// TwinCAT 3 PLC project PLC
// ProgramVersion: 3.1.4024.0
// libraries:
//   CmpBitmapPool, * (System)
//   Tc2_Standard, * (Beckhoff Automation GmbH)
//   Tc2_System, * (Beckhoff Automation GmbH)
//   Tc3_Module, * (Beckhoff Automation GmbH)
//   VisuDialogs, * (System)
//   VisuSymbols,3.5.10.0,System
// project tree:
//   DUTs/ DPLC.TcPOU
//   / GlobalTextList.TcGTLO, ImagePool.TcIPO (not stored), PlcTask.TcTTO, VisualizationManager.TcVMO (not stored), VISU_TASK.TcTTO
//   GVLs/ GVL.TcGVL
//   POUs/ Drive_Communication.TcPOU, Hour_Meter.TcPOU, Imperial_Metric_Switching.TcPOU, Pelletizer_Speed_Control.TcPOU, Pellet_Calibration.TcPOU
//   VISUs/ Calculations_Settings.TcVIS, Machine_ID_Settings.TcVIS, Calibrate_Settings.TcVIS, Rotor_Settings.TcVIS, Preset_Pellet_Length.TcVIS, Feedroll_Settings.TcVIS, Home.TcVIS, Settings_Menu.TcVIS
// real-time tasks:
//   TASK PlcTask: cycle T#3ms, priority 4, ADS port 350
//   TASK VISU_TASK: cycle T#200000us, priority 30, ADS port 351
// I/O:
//   DEVICE Device 1 (EtherCAT) (disabled), AmsNetId 10.0.1.31.2.1
//     Feedroll Drive(Inverter i550 Cabinet) [i550 Cabinet V07.00.xx] (disabled)
//     Rotor Drive(Inverter i550 Cabinet) [i550 Cabinet V06.04.xx] (disabled)
// variable links:
//   PLC/PLC Instance <-> Device 1 (EtherCAT)/Feedroll Drive(Inverter i550 Cabinet)
//     PlcTask Inputs/Drive_Communication.Feedroll_Drive_Running <-> TPDO (A) user config/NetWordOUT1 @bit 6
//     PlcTask Inputs/GVL.Actual_FeedrollMot_Speed_RPM <-> TPDO (A) Velocity/Actual speed
//     PlcTask Inputs/GVL.FeedrolAnalogInput <-> TPDO (A) user config/feedrollanaloginput1
//     PlcTask Outputs/Pelletizer_Speed_Control.FeedrollMot_Speed_Hz <-> RPDO (A) user config/Velocity mode setpoint
//   PLC/PLC Instance <-> Device 1 (EtherCAT)/Rotor Drive(Inverter i550 Cabinet)
//     PlcTask Inputs/Drive_Communication.Rotor_Active_Torque <-> TPDO (A) user config/Actual torque
//     PlcTask Inputs/Drive_Communication.Rotor_Drive_Running <-> TPDO (A) user config/NetWordOUT1 @bit 6
//     PlcTask Inputs/GVL.Actual_RotorMot_Speed_RPM <-> TPDO (A) Velocity/Actual speed
//     PlcTask Outputs/Pelletizer_Speed_Control.RotorMot_Speed_Hz <-> RPDO (A) user config/Velocity mode setpoint

CONFIGURATION PLC
    RESOURCE PLC ON TwinCAT3
        TASK PlcTask(INTERVAL := T#3ms, PRIORITY := 4);
        TASK VISU_TASK(INTERVAL := T#200000us, PRIORITY := 30);
        PROGRAM Pelletizer_Speed_Control WITH PlcTask : Pelletizer_Speed_Control;
        PROGRAM Drive_Communication WITH PlcTask : Drive_Communication;
        PROGRAM Pellet_Calibration WITH PlcTask : Pellet_Calibration;
        PROGRAM Imperial_Metric_Switching WITH PlcTask : Imperial_Metric_Switching;
        PROGRAM Hour_Meter WITH PlcTask : Hour_Meter;
        PROGRAM VisuElems_Visu_Prg WITH VISU_TASK : VisuElems.Visu_Prg;
    END_RESOURCE
END_CONFIGURATION

// ---- GVLs/GVL.TcGVL
{attribute 'qualified_only'}
VAR_GLOBAL


////////////////////////////////////////////////////////////////////////////////////
////////////////////////////////////////Pelletizer Control I/O /////////////////////

/////////////////Start/Stop
//Start : BOOL;
//Stop : BOOL;
//Running: BOOL;
/////////////////////////////
//Not using Start and Stop bits for the Normal DPLC Program, if start and stop buttons were on the screen, we would use them.

/////////////////Feedroll Control
Feedroll_Set_RPM : REAL;
FeedRate_Line_Speed : REAL;
Feedroll_Calculated_RPM : REAL;
Actual_FeedrollMot_Speed_RPM AT %I* : INT;
/////////////////////////////

/////////////////Rotor Control
Rotor_Calculated_RPM : REAL;
Rotor_RPMLimit_Exceeded : REAL; 
Rotor_RPM_Minimum : REAL;
Actual_RotorMot_Speed_RPM AT %I* : INT;
/////////////////////////////

/////////////////Machine Control
Speed_Input : REAL;
FeedrolAnalogInput  AT %I*: INT;	//Analog Input as a percentage of the Analog Input Setting // 0-10V__0-100%
Pellet_Length_Output : REAL;
Pelletizer_Running :BOOL;
Rotor_Drive_Fault : BOOL;
Feedroll_Drive_Fault: BOOL;
//Safety
Cover_Open : BOOL;
Emergency_Stop_Active : BOOL;
Discharge_Chute_NotPresent : BOOL;
/////////////////////////////

////////////////Calculated Data 
Minimum_Pellet_Length : REAL;
Maximum_Pellet_Length : REAL;
Minimum_Line_Speed : REAL;
Maximum_Line_Speed : REAL;
/////////////////////////////
END_VAR


VAR_GLOBAL PERSISTENT
///PERSISTENT VARIABLES: retain their value after an uncontrolled termination, a Reset cold or a new download of the PLC project. 
	Machine_Serial_Number : STRING;
	Electrical_Bill_ID : STRING;
	Purchase_Order_Number : STRING;
	Work_Order_Number : STRING;
	
///////////////////////////////////////////////////////////////////////////////////////
////////////////////////////////Pelletizer Setup Data//////////////////////////////////

////////////////Rotor Motor Data
RotorMot_Rated_Hz : REAL;
RotorMot_Rated_RPM : REAL;
RotorMot_Max_Hz : REAL;
RotorMot_Min_Hz : REAL;
RotorMot_Measured_60Hz_RPM : REAL;
///////////////////////////////

/////////////////////Rotor Data
Rotor_Tooth_Count : REAL;
Rotor_RPM_Limit : REAL;
Rotor_Drive_Pulley : REAL;
Rotor_Driven_Pulley : REAL;
///////////////////////////////

////////////Feedroll Motor Data
FeedrollMot_Rated_RPM : REAL;
FeedrollMot_Rated_Hz : REAL;
FeedrollMot_Max_Hz : REAL;
FeedrollMot_Min_Hz : REAL;
//////////////////////////////

/////////////////Feedroll Data
Feedroll_Diameter_Inch : REAL;
Feedroll_Drive_Pulley : REAL;
Feedroll_Driven_Pulley : REAL;
Feedroll_Pressure : REAL;
/////////////////////////////

////////////////////////Misc
Metric_Set_Bit : BOOL;
Preset1 : REAL := 0.125;
Preset2 : REAL := 0.118;
Preset3 : REAL := 0.100;
Preset4 : REAL := 0.088;
//////////////////////////////

//////////////////////////Calibration
Pellet_Length_Calibration_Value : REAL := 1;
Pellet_Length_Inch_Input : REAL;
//////////////////////////////////////
END_VAR

// ---- POUs/Pelletizer_Speed_Control.TcPOU
PROGRAM Pelletizer_Speed_Control
VAR
	FirstScan : BOOL := TRUE;
	TempSpeed: REAL;
	
	FeedrollMot_Speed_Hz AT %Q*: INT;	//Map to Drive Parameter for Speed control Using Hertz
	RotorMot_Speed_Hz  AT %Q*: INT;		//Map to Drive Parameter for Speed control Using Hertz
	
END_VAR

//Read Analog Input for speed setting as Percentage.
TempSpeed := INT_TO_REAL(GVL.FeedrolAnalogInput) / 1000;


IF GVL.Pelletizer_Running OR FirstScan THEN
	
DPLC(
	Pellet_Length_Inch_Input := Imperial_Metric_Switching.Pellet_Length_Imperial_Input, 
	Speed_Input := 	TempSpeed, 
	RotorMot_Rated_RPM := GVL.RotorMot_Measured_60Hz_RPM, 
	RotorMot_Rated_Hz := GVL.RotorMot_Rated_Hz, 
	RotorMot_Max_Hz := GVL.RotorMot_Max_Hz,
	RotorMot_Min_Hz := GVL.RotorMot_Min_Hz,
	Rotor_Drive_Pulley := GVL.Rotor_Drive_Pulley,
	Rotor_Driven_Pulley := GVL.Rotor_Driven_Pulley, 
	Rotor_Tooth_Count := GVL.Rotor_Tooth_Count, 
	Rotor_RPM_Limit := GVL.Rotor_RPM_Limit,
	FeedrollMot_Rated_RPM := GVL.FeedrollMot_Rated_RPM, 
	FeedrollMot_Rated_Hz := GVL.FeedrollMot_Rated_Hz, 
	FeedrollMot_Max_Hz := GVL.FeedrollMot_Max_Hz,
	FeedrollMot_Min_Hz := GVL.FeedrollMot_Min_Hz,
	Actual_FeedrollMot_Speed_RPM := GVL.Actual_FeedrollMot_Speed_RPM,
	Feedroll_Drive_Pulley := GVL.Feedroll_Drive_Pulley, 
	Feedroll_Driven_Pulley := GVL.Feedroll_Driven_Pulley, 
	Feedroll_Diameter_Inch := GVL.Feedroll_Diameter_Inch, 
	Metric_Set_Bit := GVL.Metric_Set_Bit,
	Pellet_Length_Output => GVL.Pellet_Length_Output,
	Feedroll_Motor_Speed_Hz_int => Pelletizer_Speed_Control.FeedrollMot_Speed_Hz, 
	Rotor_Motor_Speed_Hz_int => Pelletizer_Speed_Control.RotorMot_Speed_Hz,
	Rotor_Speed_RPM => GVL.Rotor_Calculated_RPM,
	FeedRate_Feet_Per_Minute => GVL.FeedRate_Line_Speed,
	Rotor_RPM_Minimum => GVL.Rotor_RPM_Minimum,
	Maximum_Line_Speed => GVL.Maximum_Line_Speed,
	Minimum_Line_Speed => GVL.Minimum_Line_Speed,
	Maximum_Pellet_Length => GVL.Maximum_Pellet_Length,
	Minimum_Pellet_Length => GVL.Minimum_Pellet_Length
);

ELSE
	GVL.Rotor_Calculated_RPM := 0;//Display 0 when not running.
	GVL.FeedRate_Line_Speed := 0;//Display 0 when not running.
END_IF

FirstScan := FALSE;

END_PROGRAM

// ---- DUTs/DPLC.TcPOU
FUNCTION DPLC : REAL
VAR_INPUT
	Pellet_Length_Inch_Input :REAL;
	Speed_Input: REAL;	//The speed input must be a percentage.

	RotorMot_Rated_RPM : REAL;
	RotorMot_Rated_Hz: REAL;
	RotorMot_Max_Hz : REAL;
	RotorMot_Min_Hz : REAL;

	Rotor_Drive_Pulley: REAL;
	Rotor_Driven_Pulley: REAL;
	Rotor_Tooth_Count: REAL;
	Rotor_RPM_Limit: REAL;
	
	FeedrollMot_Rated_RPM: REAL;
	FeedrollMot_Rated_Hz: REAL;
	FeedrollMot_Max_Hz : REAL;
	FeedrollMot_Min_Hz : REAL;
	Actual_FeedrollMot_Speed_RPM : INT;

	Feedroll_Drive_Pulley: REAL;
	Feedroll_Driven_Pulley: REAL;
	Feedroll_Diameter_Inch: REAL;
	

	Metric_Set_Bit : BOOL;

END_VAR

VAR
	FeedrollMot_Speed_Hz : REAL;
	FeedrollMot_Speed_RPM : REAL;
	FeedrollMot_RPM_Per_Hz : REAL;

	Feedroll_Pulley_Ratio: REAL;
	Feedroll_Speed_RPM: REAL;
	Feedroll_Circumference_Inch :REAL;

	RotorMot_Speed_Hz : REAL;
	RotorMot_Speed_RPM : REAL;
	RotorMot_RPM_Per_Hz : REAL;

	Rotor_Pulley_Ratio: REAL;
	Cuts_Per_Minute: REAL;
	
	Min_Cuts_Per_Minute : REAL;
	Max_Cuts_Per_Minute : REAL;
	
	FeedRate_Inches_Per_Minute: REAL;
END_VAR

VAR_OUTPUT
	Pellet_Length_Output :REAL; 		//this is the resulting pellet length for display. Converted to Metric or Imperial depending on the Metric Set Bit.

	Feedroll_Motor_Speed_Hz_int : INT;	//this variable is written to the drive. Ms: Velocity Mode (-2) uses Hz to control speed.
	Rotor_Motor_Speed_Hz_int : INT;  	//this variable is written to the drive. Ms: Velocity Mode (-2) uses Hz to control speed.
	
	Rotor_Speed_RPM: REAL;
	
	FeedRate_Feet_Per_Minute: REAL;		//This is the displayed Ft/min on the HMI
	
	Rotor_RPM_Minimum : REAL; // info for Gauge on HMI
	Maximum_Line_Speed : REAL;	//info for machine limits
	Minimum_Line_Speed: REAL;	//info for machine limits
	Maximum_Pellet_Length : REAL;	//info for machine limits
	Minimum_Pellet_Length : REAL;	//info for machine limits
END_VAR

////////////////////////////Notes and Information/////////////////////////////////////////////////////////////////////////////////////////////////////
//         The feedroll Must be the master for the DPLC calculations
//         The reason for this is so that the line speed can be set BEFORE the pellet length is determined
//         When actively changing the pellet length while running, the rotor speed can change but the feedrate must be maintained.
//////////////////////////////////////////////////////////////////////////////////////////////////////////////////////////////////////////////////////
//If the Metric Bit is set, we convert the pellet length in mm to inches for input. We also convert to output Feedroll speed to meters per minute

//if direction is backwards, make it a postive number.
IF Actual_feedrollMot_Speed_RPM < 0 THEN
	Actual_feedrollMot_Speed_RPM := Actual_feedrollMot_Speed_RPM * -1;
END_IF
	


////////////////////////////////////Setup Calculations
FeedrollMot_RPM_Per_Hz := FeedrollMot_Rated_RPM / FeedrollMot_Rated_Hz;
Feedroll_Pulley_Ratio := Feedroll_Drive_Pulley / Feedroll_Driven_Pulley;
Feedroll_Circumference_Inch := Feedroll_Diameter_Inch *  3.14159;

RotorMot_RPM_Per_Hz := RotorMot_Rated_RPM / RotorMot_Rated_Hz;	
Rotor_Pulley_Ratio := Rotor_Drive_Pulley / Rotor_Driven_pulley;


/////////////////////////////////////Feedroll Calculations
FeedrollMot_Speed_Hz := FeedrollMot_Max_Hz * Speed_Input;
FeedrollMot_Speed_RPM := INT_TO_REAL(Actual_FeedrollMot_Speed_RPM);	// Read the Feedroll RPM Back and do calculation on the actual.
Feedroll_Speed_RPM := FeedrollMot_Speed_RPM * Feedroll_Pulley_Ratio;
FeedRate_Inches_Per_Minute := Feedroll_Speed_RPM * Feedroll_Circumference_Inch;
FeedRate_Feet_Per_Minute := FeedRate_Inches_Per_Minute / 12 ;


/////////////////////////////////////Rotor Calculations
Cuts_Per_Minute := FeedRate_Inches_Per_Minute / (Pellet_Length_Inch_Input * GVL.Pellet_Length_Calibration_Value);
Rotor_Speed_RPM := Cuts_Per_Minute / Rotor_Tooth_Count;	//the ROTOR needs to go this many RPM to achieve the pellet length
RotorMot_Speed_RPM := Rotor_Speed_RPM / Rotor_Pulley_Ratio;
RotorMot_Speed_Hz := RotorMot_Speed_RPM / RotorMot_RPM_Per_Hz;


////////////////////////////////////Set and Convert Speeds to send to Drive
Feedroll_Motor_Speed_Hz_int := REAL_TO_INT(FeedrollMot_Speed_Hz * 10);
Rotor_Motor_Speed_Hz_int := REAL_TO_INT(RotorMot_Speed_Hz * 10);


///////////////////////////////////Limits
Maximum_Line_Speed := (Feedroll_Circumference_Inch / 12) * ((FeedrollMot_Max_Hz * FeedrollMot_RPM_Per_Hz) * Feedroll_Pulley_Ratio);
Minimum_Line_Speed := (Feedroll_Circumference_Inch / 12) * ((FeedrollMot_Min_Hz * FeedrollMot_RPM_Per_Hz) * Feedroll_Pulley_Ratio);

Rotor_RPM_Minimum := RotorMot_RPM_Per_Hz * RotorMot_Min_Hz;

Min_Cuts_Per_Minute := Rotor_Tooth_Count * ((RotorMot_RPM_Per_Hz * RotorMot_Min_Hz) * Rotor_Pulley_Ratio);
Max_Cuts_Per_Minute := Rotor_Tooth_Count * ((RotorMot_RPM_Per_Hz * RotorMot_Max_Hz) * Rotor_Pulley_Ratio);

Maximum_Pellet_Length := (Maximum_Line_Speed * 12) / Min_Cuts_Per_Minute;
Minimum_Pellet_Length := (Minimum_Line_Speed * 12) / Max_Cuts_Per_Minute;


IF Metric_Set_Bit THEN
	//Convert feedroll speed to meters per min for display.
	Feedrate_Feet_Per_Minute := Feedrate_Feet_Per_Minute * 0.3048;
	Maximum_Line_Speed := Maximum_Line_Speed * 0.3048;
	Minimum_Line_Speed := Minimum_Line_Speed * 0.3048;
	
	//Convert min and max pellet length to mm so the input box does not error.
	Maximum_Pellet_Length := Maximum_Pellet_Length * 25.4;
	Minimum_Pellet_Length := Minimum_Pellet_Length * 25.4;
END_IF

END_FUNCTION

// ---- POUs/Imperial_Metric_Switching.TcPOU
PROGRAM Imperial_Metric_Switching
VAR PERSISTENT
	Pellet_Length_Displayed : REAL;
	Pellet_Length_Metric_Input : REAL;
	Pellet_Length_Imperial_Input : REAL;
END_VAR



IF GVL.Metric_Set_Bit THEN
		Pellet_Length_Displayed := Pellet_Length_Metric_Input;
		Pellet_Length_Imperial_Input := Pellet_Length_Metric_Input / 25.4;
ELSE
		Pellet_Length_Displayed := Pellet_Length_Imperial_Input;
		Pellet_Length_Metric_Input := Pellet_Length_Imperial_Input * 25.4;
END_IF

END_PROGRAM

// ---- POUs/Drive_Communication.TcPOU
PROGRAM Drive_Communication
VAR
	Rotor_Active_Torque AT %I*: INT;	//Rotor Torque as percentage of Rated Motor Torque
	Rotor_Active_Torque_REAL : REAL;
	Rotor_Displayed_Torque :REAL;

	//Feedroll Drive
	Feedroll_Drive_Message AT %I* : USINT;		//Drive Faults
	Feedroll_Drive_Status AT %I* : UINT;
	Feedroll_Drive_Running AT %I* : BOOL;

	
	
	//Rotor Drive
	Rotor_Drive_Message AT %I* : USINT;		//Drive Faults
	Rotor_Drive_Status AT %I* : UINT;
	Rotor_Drive_Running AT %I* : BOOL;


	
	
END_VAR


/////////////////////////Rotor Torque Display Scaling
IF Rotor_Active_Torque < 0 THEN
	Rotor_Active_Torque := Rotor_Active_Torque * -1;
END_IF
Rotor_Active_Torque_REAL := INT_TO_REAL(Rotor_Active_Torque);
Rotor_Displayed_Torque := Rotor_Active_Torque_REAL / 10;



////////////////////////////////////Combined Running Status
IF Feedroll_Drive_Running AND Rotor_Drive_Running THEN
	GVL.Pelletizer_Running := TRUE;
ELSE
	GVL.Pelletizer_Running := FALSE;
END_IF

END_PROGRAM

// ---- POUs/Pellet_Calibration.TcPOU
PROGRAM Pellet_Calibration
VAR
	SET_CALIBRATON_VALUE : BOOL;
	Pellet_Length_Measured_Input : REAL;
	Pellet_Length_Temp_Cal_Val : REAL;
END_VAR

 Pellet_Length_Temp_Cal_Val :=  GVL.Pellet_Length_Inch_Input / Pellet_Length_Measured_Input;


IF SET_CALIBRATON_VALUE THEN
	GVL.Pellet_Length_Calibration_Value := Pellet_Length_Temp_Cal_Val; //this line is run by the Visu when the button is pressed.
END_IF

END_PROGRAM

// ---- POUs/Hour_Meter.TcPOU
PROGRAM Hour_Meter
VAR PERSISTENT
  	MyTimer   : TON;
	TempRun: BOOL;
END_VAR
VAR PERSISTENT
	TotalHours : REAL;
	TotalMinutes : REAL;
END_VAR

MyTimer(IN := TempRun, PT := T#1M);

IF GVL.Pelletizer_Running THEN
	TempRun:= TRUE;
END_IF

IF MyTimer.Q THEN
	TotalMinutes := TotalMinutes + 1;
	TotalHours := TotalHours + (1 / 60);
	TempRun := FALSE;
END_IF


IF TotalMinutes >= 60 THEN
	TotalHours := TotalHours + 1;	
	TotalMinutes := 0;
END_IF

END_PROGRAM

// ---- GlobalTextList.TcGTLO
TEXTLIST GlobalTextList
  548 = '%1.3f'
  110 = '%1.3F'
  99 = '%1.4f'
  937 = '%1.4F'
  640 = '%d'
  190 = '%f'
  605 = '%i'
  556 = '%s'
  3 = '0.08'
  952 = '0.088'
  997 = '0.100'
  829 = '0.125'
  500 = '0.2'
  759 = '0.200'
  928 = 'Admin'
  934 = 'Calculated Data'
  250 = 'Calibrate Pellet Length'
  455 = 'Electrical Bill ID'
  380 = 'Feedroll Data'
  838 = 'Feedroll Diameter (Inch)'
  98 = 'Feedroll Drive Pulley'
  346 = 'Feedroll Driven Pulley'
  345 = 'Feedroll Motor Data'
  241 = 'Feedroll Motor Max Hz'
  84 = 'Feedroll Motor Rated Hz'
  338 = 'Feedroll Motor Rated RPM'
  989 = 'Feedroll Speed'
  549 = 'Ft/Min'
  818 = 'Hour Meter'
  310 = 'Hours'
  753 = 'Inch             mm'
  420 = 'Limits'
  892 = 'Login'
  925 = 'Machine Identity'
  220 = 'Maximum Pellet Length'
  970 = 'Maximum Rated Line Speed'
  923 = 'Maximum Rated Line Speed (Ft/min)'
  263 = 'Minimum Feedroll Hz'
  541 = 'Minimum Feedroll Motor Hz'
  957 = 'Minimum Pellet Length'
  381 = 'Minimum Rated Line Speed'
  750 = 'Minimum Rotor Motor Hz'
  820 = 'None'
  538 = 'Operator'
  100 = 'Pellet Length'
  698 = 'Pellet Length Calibration Factor'
  471 = 'Pellet Length Measured (Actual Length)'
  815 = 'Pellet Length Setting (current setting)'
  347 = 'Pellet Length Setting (Current Setting)'
  983 = 'Preset 1'
  795 = 'Preset 2'
  126 = 'Preset 3'
  670 = 'Preset 4'
  800 = 'Purchase Order #'
  81 = 'Rotor Data'
  592 = 'Rotor Drive Pulley'
  173 = 'Rotor Driven Pulley'
  584 = 'Rotor Motor Data'
  294 = 'Rotor Motor Max Hz'
  29 = 'Rotor Motor Rated Hz'
  624 = 'Rotor Motor Rated RPM'
  597 = 'Rotor Speed'
  528 = 'Rotor Tooth Count'
  903 = 'Rotor Torque Percent'
  867 = 'Rotor Torque Utilization %'
  770 = 'RPM'
  105 = 'Serial Number'
  733 = 'Service'
  324 = 'Work Order #'
  850 = 'Wr'
  139 = 'WRITE CALIBRATION CONSTANT'
END_TEXTLIST

// ---- VISUs/Calculations_Settings.TcVIS
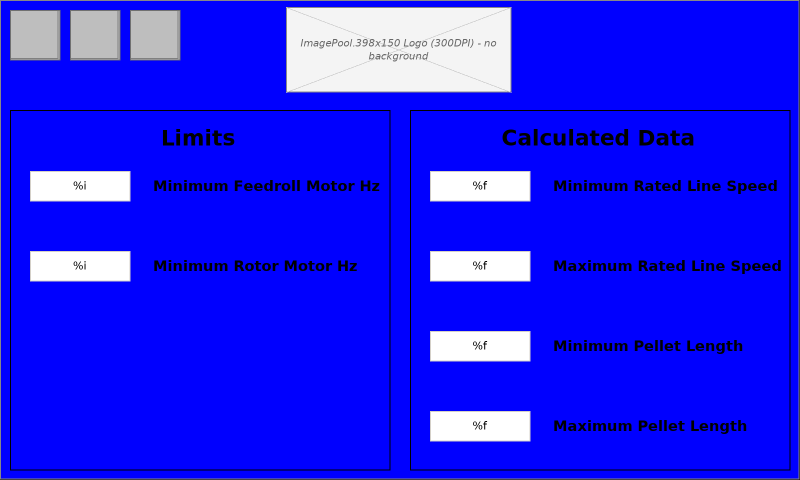
VISUALIZATION Calculations_Settings  // 800x480
    Rectangle (0,0 800x480)
    Rectangle (10,110 380x360)
    Textfield (30,171 100x30), "%i", text variable: GVL.FeedrollMot_Min_Hz
        OnMouseClick: write the text variable via VisuDialogs.Numpad
    Rectangle (410,110 380x360)
    Textfield (30,251 100x30), "%i", text variable: GVL.RotorMot_Min_Hz
        OnMouseClick: write the text variable via VisuDialogs.Keypad
    Textfield (430,411 100x30), "%f", text variable: GVL.Maximum_Pellet_Length
    Image (286,7 225x85), image: ImagePool.398x150 Logo (300DPI) - no background
        OnMouseClick: change screen: Home
    Button (70,10 50x50), image: VisuSymbols.Symbols.Home
        OnMouseClick: change screen: Home
    Label (20,120 357x36), "Limits"
    Label (420,120 357x36), "Calculated Data"
    Button (10,10 50x50), image: VisuSymbols.Symbols.TriangleLeft
        OnMouseClick: change screen: Previous Home
    Textfield (430,171 100x30), "%f", text variable: GVL.Minimum_Line_Speed
    Textfield (430,251 100x30), "%f", text variable: GVL.Maximum_Line_Speed
    Textfield (430,331 100x30), "%f", text variable: GVL.Minimum_Pellet_Length
    Label (150,171 225x30), "Minimum Feedroll Motor Hz"
    Label (150,251 225x30), "Minimum Rotor Motor Hz"
    Label (550,411 225x30), "Maximum Pellet Length"
    Label (550,171 225x30), "Minimum Rated Line Speed"
    Label (550,251 237x30), "Maximum Rated Line Speed"
    Label (550,331 225x30), "Minimum Pellet Length"
    Button (130,10 50x50), image: VisuSymbols.Symbols.TwoWheels
        OnMouseClick: change screen: Settings_Menu
END_VISUALIZATION

// ---- VISUs/Machine_ID_Settings.TcVIS
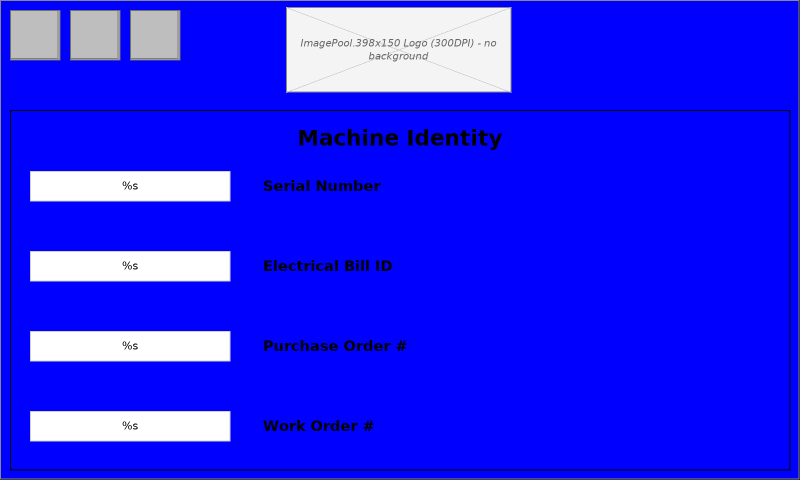
VISUALIZATION Machine_ID_Settings  // 800x480
    Rectangle (0,0 800x480)
    Rectangle (10,110 780x360)
    Textfield (30,171 200x30), "%s", text variable: GVL.Machine_Serial_Number
        OnMouseClick: write the text variable via VisuDialogs.Keypad
    Textfield (30,251 200x30), "%s", text variable: GVL.Electrical_Bill_ID
        OnMouseClick: write the text variable via VisuDialogs.Keypad
    Textfield (30,331 200x30), "%s", text variable: GVL.Purchase_Order_Number
        OnMouseClick: write the text variable via VisuDialogs.Keypad
    Image (286,7 225x85), image: ImagePool.398x150 Logo (300DPI) - no background
        OnMouseClick: change screen: Home
    Button (70,10 50x50), image: VisuSymbols.Symbols.Home
        OnMouseClick: change screen: Home
    Label (0,120 800x36), "Machine Identity"
    Button (10,10 50x50), image: VisuSymbols.Symbols.TriangleLeft
        OnMouseClick: change screen: Previous Home
    Textfield (30,411 200x30), "%s", text variable: GVL.Work_Order_Number
        OnMouseClick: write the text variable via VisuDialogs.Keypad
    Label (260,171 225x30), "Serial Number"
    Label (260,251 225x30), "Electrical Bill ID"
    Label (260,331 225x30), "Purchase Order #"
    Label (260,411 225x30), "Work Order #"
    Label (550,331 225x30)
    Button (130,10 50x50), image: VisuSymbols.Symbols.TwoWheels
        OnMouseClick: change screen: Settings_Menu
END_VISUALIZATION

// ---- VISUs/Calibrate_Settings.TcVIS
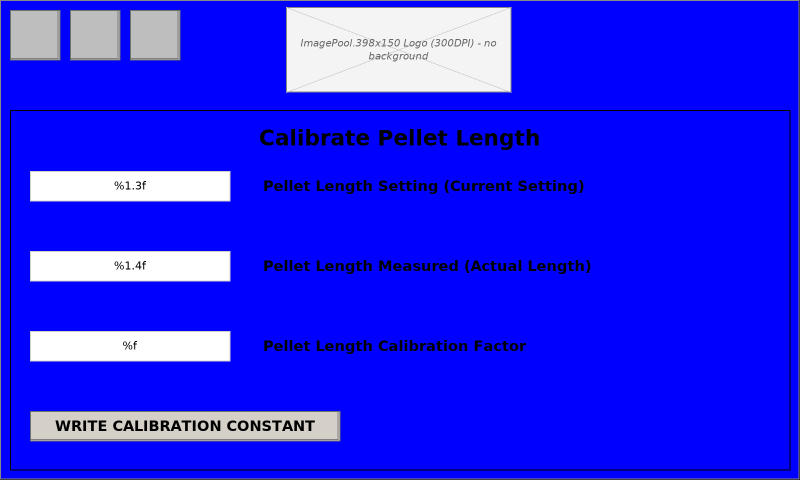
VISUALIZATION Calibrate_Settings  // 800x480
    Rectangle (0,0 800x480)
    Rectangle (10,110 780x360)
    Textfield (30,171 200x30), "%1.3f", text variable: GVL.Pellet_Length_Inch_Input
    Textfield (30,251 200x30), "%1.4f", text variable: Pellet_Calibration.Pellet_Length_Measured_Input
        OnMouseClick: write the text variable via VisuDialogs.Numpad
    Textfield (30,331 200x30), "%f", text variable: Pellet_Calibration.Pellet_Length_Temp_Cal_Val
    Image (286,7 225x85), image: ImagePool.398x150 Logo (300DPI) - no background
        OnMouseClick: change screen: Home
    Button (70,10 50x50), image: VisuSymbols.Symbols.Home
        OnMouseClick: change screen: Home
    Label (0,120 800x36), "Calibrate Pellet Length"
    Button (10,10 50x50), image: VisuSymbols.Symbols.TriangleLeft
        OnMouseClick: change screen: Previous Home
    Label (260,171 361x30), "Pellet Length Setting (Current Setting)"
    Label (260,251 421x30), "Pellet Length Measured (Actual Length)"
    Label (260,331 322x30), "Pellet Length Calibration Factor"
    Label (260,411 225x30)
    Label (550,331 225x30)
    Button (30,411 310x30), "WRITE CALIBRATION CONSTANT", pressed state: Pellet_Calibration.SET_CALIBRATON_VALUE
        OnMouseClick: execute { GVL.Pellet_Length_Calibration_Value := Pellet_Calibration.Pellet_Length_Temp_Cal_Val; }
    Button (130,10 50x50), image: VisuSymbols.Symbols.TwoWheels
        OnMouseClick: change screen: Settings_Menu
END_VISUALIZATION

// ---- VISUs/Rotor_Settings.TcVIS
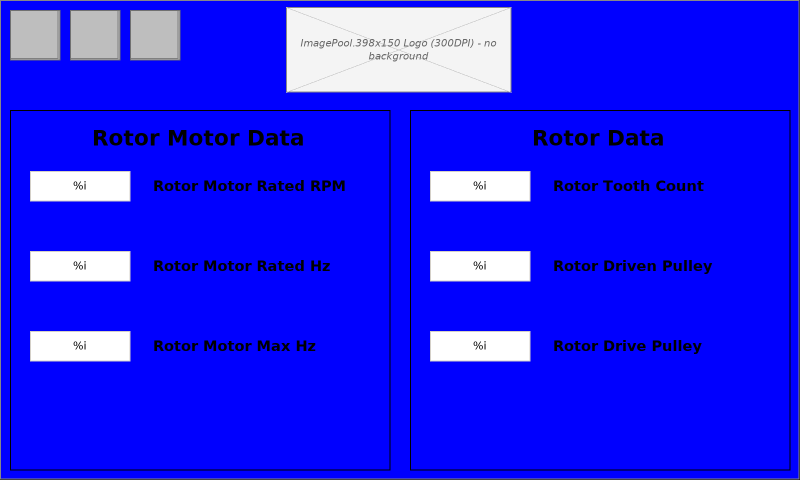
VISUALIZATION Rotor_Settings  // 800x480
    Rectangle (0,0 800x480)
    Rectangle (10,110 380x360)
    Textfield (30,171 100x30), "%i", text variable: GVL.RotorMot_Rated_RPM
        OnMouseClick: write the text variable via VisuDialogs.Numpad
    Rectangle (410,110 380x360)
    Textfield (30,251 100x30), "%i", text variable: GVL.RotorMot_Rated_Hz
        OnMouseClick: write the text variable via VisuDialogs.Numpad
    Textfield (30,331 100x30), "%i", text variable: GVL.RotorMot_Max_Hz
        OnMouseClick: write the text variable via VisuDialogs.Numpad
    Image (286,7 225x85), image: ImagePool.398x150 Logo (300DPI) - no background
        OnMouseClick: change screen: Home
    Button (70,10 50x50), image: VisuSymbols.Symbols.Home
        OnMouseClick: change screen: Home
    Label (20,120 357x36), "Rotor Motor Data"
    Label (420,120 357x36), "Rotor Data"
    Button (10,10 50x50), image: VisuSymbols.Symbols.TriangleLeft
        OnMouseClick: change screen: Previous Home
    Textfield (430,171 100x30), "%i", text variable: GVL.Rotor_Tooth_Count
        OnMouseClick: write the text variable via VisuDialogs.Numpad
    Textfield (430,251 100x30), "%i", text variable: GVL.Rotor_Driven_Pulley
        OnMouseClick: write the text variable via VisuDialogs.Numpad
    Textfield (430,331 100x30), "%i", text variable: GVL.Rotor_Drive_Pulley
        OnMouseClick: write the text variable via VisuDialogs.Numpad
    Label (150,171 225x30), "Rotor Motor Rated RPM"
    Label (150,251 225x30), "Rotor Motor Rated Hz"
    Label (150,331 225x30), "Rotor Motor Max Hz"
    Label (550,171 225x30), "Rotor Tooth Count"
    Label (550,251 225x30), "Rotor Driven Pulley"
    Label (550,331 225x30), "Rotor Drive Pulley"
    Button (130,10 50x50), image: VisuSymbols.Symbols.TwoWheels
        OnMouseClick: change screen: Settings_Menu
END_VISUALIZATION

// ---- VISUs/Preset_Pellet_Length.TcVIS
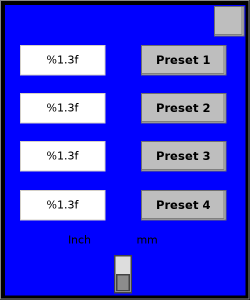
VISUALIZATION Preset_Pellet_Length  // 250x300
    Rectangle (0,0 250x300)
    Textfield (20,45 85x30), "%1.3f", text variable: GVL.Preset1
        OnMouseClick: write the text variable via VisuDialogs.Numpad
    Textfield (20,93 85x30), "%1.3f", text variable: GVL.Preset2
        OnMouseClick: write the text variable via VisuDialogs.Numpad
    Textfield (20,141 85x30), "%1.3f", text variable: GVL.Preset3
        OnMouseClick: write the text variable via VisuDialogs.Numpad
    Textfield (20,190 85x30), "%1.3f", text variable: GVL.Preset4
        OnMouseClick: write the text variable via VisuDialogs.Numpad
    DipSwitch (82,255 82x38), variable: GVL.Metric_Set_Bit, behaviour: TOGGLE, style: Switch-DipSwitch-Gray
    Label (38,225 150x30), "Inch mm"
    Button (141,93 85x30), "Preset 2", text variable: GVL.Preset2
        OnMouseClick: execute {
            IF GVL.Metric_Set_Bit THEN
            	Imperial_Metric_Switching.Pellet_Length_Metric_Input := GVL.Preset2;
            ELSE
            	Imperial_Metric_Switching.Pellet_Length_Imperial_Input := GVL.Preset2;
            END_IF
        }
    Button (141,45 85x30), "Preset 1"
        OnMouseClick: execute {
            IF GVL.Metric_Set_Bit THEN
            	Imperial_Metric_Switching.Pellet_Length_Metric_Input := GVL.Preset1;
            ELSE
            	Imperial_Metric_Switching.Pellet_Length_Imperial_Input := GVL.Preset1;
            END_IF
        }
    Button (141,141 85x30), "Preset 3", text variable: GVL.Preset3
        OnMouseClick: execute {
            IF GVL.Metric_Set_Bit THEN
            	Imperial_Metric_Switching.Pellet_Length_Metric_Input := GVL.Preset3;
            ELSE
            	Imperial_Metric_Switching.Pellet_Length_Imperial_Input := GVL.Preset3;
            END_IF
        }
    Button (141,190 85x30), "Preset 4", text variable: GVL.Preset4
        OnMouseClick: execute {
            IF GVL.Metric_Set_Bit THEN
            	Imperial_Metric_Switching.Pellet_Length_Metric_Input := GVL.Preset4;
            ELSE
            	Imperial_Metric_Switching.Pellet_Length_Imperial_Input := GVL.Preset4;
            END_IF
        }
    Button (214,6 30x30), image: VisuSymbols.Symbols.Wrong
        OnMouseClick: CloseDialog Dialog=Preset_Pellet_Length, Result=None, NumpadKeypadSet=True
END_VISUALIZATION

// ---- VISUs/Feedroll_Settings.TcVIS
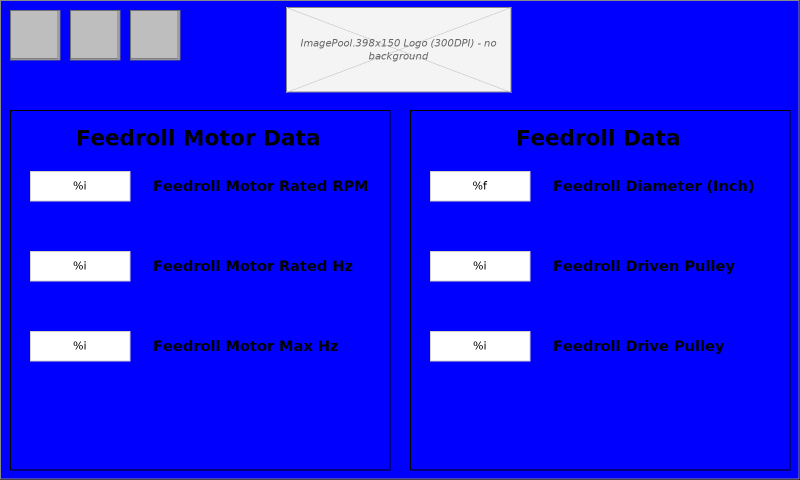
VISUALIZATION Feedroll_Settings  // 800x480
    Rectangle (0,0 800x480)
    Rectangle (10,110 380x360)
    Textfield (30,171 100x30), "%i", text variable: GVL.FeedrollMot_Rated_RPM
        OnMouseClick: write the text variable via VisuDialogs.Numpad
    Rectangle (410,110 380x360)
    Textfield (30,251 100x30), "%i", text variable: GVL.FeedrollMot_Rated_Hz
        OnMouseClick: write the text variable via VisuDialogs.Numpad
    Textfield (30,331 100x30), "%i", text variable: GVL.FeedrollMot_Max_Hz
        OnMouseClick: write the text variable via VisuDialogs.Numpad
    Image (286,7 225x85), image: ImagePool.398x150 Logo (300DPI) - no background
        OnMouseClick: change screen: Home
    Button (70,10 50x50), image: VisuSymbols.Symbols.Home
        OnMouseClick: change screen: Home
    Label (20,120 357x36), "Feedroll Motor Data"
    Label (420,120 357x36), "Feedroll Data"
    Button (10,10 50x50), image: VisuSymbols.Symbols.TriangleLeft
        OnMouseClick: change screen: Previous Home
    Textfield (430,171 100x30), "%f", text variable: GVL.Feedroll_Diameter_Inch
        OnMouseClick: write the text variable via VisuDialogs.Numpad
    Textfield (430,251 100x30), "%i", text variable: GVL.Feedroll_Driven_Pulley
        OnMouseClick: write the text variable via VisuDialogs.Numpad
    Textfield (430,331 100x30), "%i", text variable: GVL.Feedroll_Drive_Pulley
        OnMouseClick: write the text variable via VisuDialogs.Numpad
    Label (150,171 225x30), "Feedroll Motor Rated RPM"
    Label (150,251 225x30), "Feedroll Motor Rated Hz"
    Label (150,331 225x30), "Feedroll Motor Max Hz"
    Label (550,171 225x30), "Feedroll Diameter (Inch)"
    Label (550,251 225x30), "Feedroll Driven Pulley"
    Label (550,331 225x30), "Feedroll Drive Pulley"
    Button (130,10 50x50), image: VisuSymbols.Symbols.TwoWheels
        OnMouseClick: change screen: Settings_Menu
END_VISUALIZATION

// ---- VISUs/Home.TcVIS
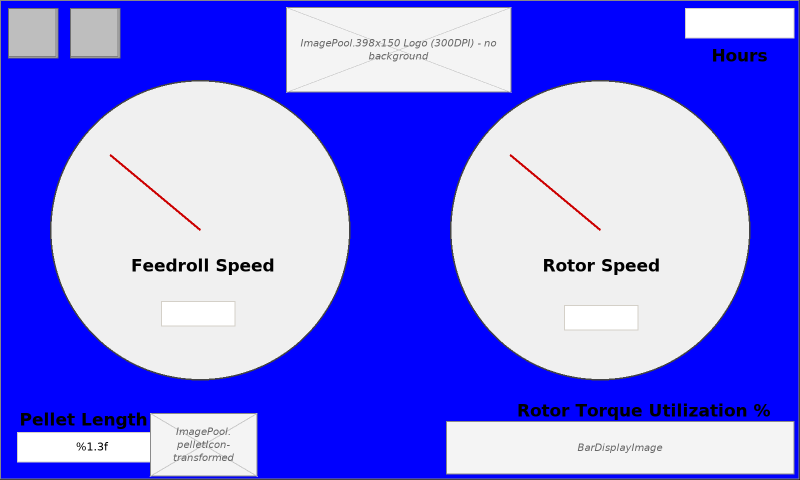
VISUALIZATION Home  // 800x480
    Rectangle (0,0 800x480)
    Meter360 (50,80 300x300), style: Meter-Meter360-Gray, scale format: %.1f, scale 0..100
        p518627256: Ft/Min
    BarDisplayImage (446,421 348x53), value: 0, style: BarDisplayImage-Gray, scale format: %.1f, scale 0..100
    Textfield (17,432 150x30), "%1.3f", text variable: Imperial_Metric_Switching.Pellet_Length_Displayed
    Textfield (161,301 74x25)
    Meter360 (450,80 300x300), style: Meter-Meter360-Gray, scale format: %.1f, scale 0..100
    Textfield (564,305 74x25)
    Image (286,7 225x85), image: ImagePool.398x150 Logo (300DPI) - no background
        OnMouseClick: change screen: Home
    Button (8,8 50x50), tooltip "Login", image: VisuSymbols.Symbols.User
        OnMouseClick: VisuUserMgmt Type=Login
    Label (685,40 109x31), "Hours"
    Textfield (685,8 109x30)
    Label (17,404 133x31), "Pellet Length"
    Label (509,395 270x31), "Rotor Torque Utilization %"
    Label (133,250 140x31), "Feedroll Speed"
    Label (535,250 133x31), "Rotor Speed"
    Button (70,8 50x50), image: VisuSymbols.Symbols.TwoWheels
        OnMouseClick: change screen: Settings_Menu
    Image (150,413 107x63), image: ImagePool.pelletIcon-transformed
        OnMouseClick: OpenDialog Dialog=Preset_Pellet_Length, OpenModal=True, OpenCentered=True
END_VISUALIZATION

// ---- VISUs/Settings_Menu.TcVIS
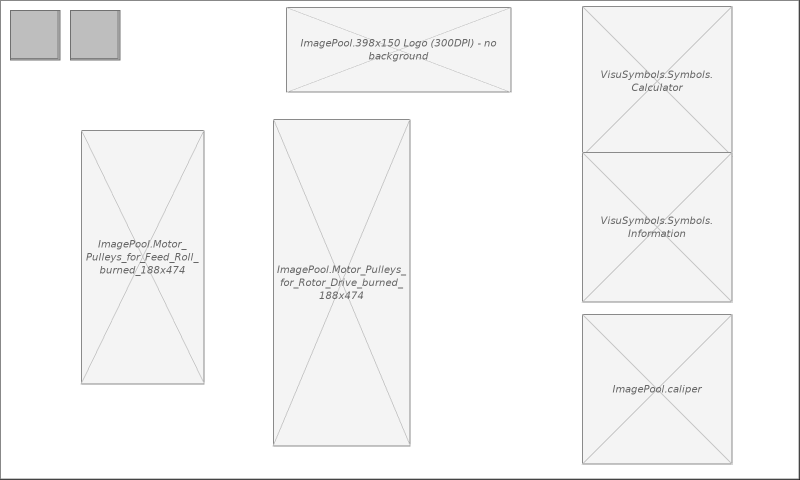
VISUALIZATION Settings_Menu  // 800x480
    Rectangle (0,0 800x480)
    Button (10,10 50x50), image: VisuSymbols.Symbols.TriangleLeft
        OnMouseClick: change screen: Previous Home
    Button (70,10 50x50), image: VisuSymbols.Symbols.Home
        OnMouseClick: change screen: Home
    Image (273,119 137x327), image: ImagePool.Motor_Pulleys_for_Rotor_Drive_burned_188x474
        OnMouseClick: change screen: Rotor_Settings
    Image (81,130 123x254), image: ImagePool.Motor_Pulleys_for_Feed_Roll_burned_188x474
        OnMouseClick: change screen: Feedroll_Settings
    Image (582,314 150x150), image: ImagePool.caliper
        OnMouseClick: change screen: Calibrate_Settings
    Image (582,6 150x150), image: VisuSymbols.Symbols.Calculator
        OnMouseClick: change screen: Calculations_Settings
    Image (582,152 150x150), image: VisuSymbols.Symbols.Information
        OnMouseClick: change screen: Machine_ID_Settings
    Image (286,7 225x85), image: ImagePool.398x150 Logo (300DPI) - no background
        OnMouseClick: change screen: Home
END_VISUALIZATION
